VISUALIZATION _VISU_GridPointView  // 120x10
VAR_IN_OUT
	m_Inst : ST_DeformationPointTbl;
END_VAR
    Rectangle (0,0 20x10), "c:%d", text variable: m_Inst.sPoint.col, colour toggle: m_Inst.bSet
    Rectangle (20,0 20x10), "r:%d", text variable: m_Inst.sPoint.row, colour toggle: m_Inst.bSet
    Rectangle (40,0 20x10), "%d", tooltip "x_ref", text variable: m_Inst.sPoint.x_ref
    Rectangle (60,0 20x10), "%d", tooltip "y_ref", text variable: m_Inst.sPoint.y_ref
    Rectangle (80,0 20x10), "%0.1f", tooltip "dx", text variable: m_Inst.sPoint.dx
    Rectangle (100,0 20x10), "%0.1f", tooltip "dy", text variable: m_Inst.sPoint.dy
    Label (12,0 10x10), "/"
END_VISUALIZATION

(* stored: Version 1.1.0.1, ProductVersion 3.1.4024.3
   Visu _VISU_GridPointView: Id {4bc97a5d-5878-4e0d-9e61-da175d6950a0} *)
